Staubli VAL3: SocketMove.dtx

mdesc mNomSpeed
string sGetStr
sio sS = {link=Socket\ss}
string sBuff
trsf trTrsf
trsf trPara
bool bRes
mdesc mRun
pointRx pPrun = {fatherId=world[0]}
tool tTool = {z=100, fatherId=flange[0], ioLink=valve1}
jointRx jrun
pointRx pPMovec = {fatherId=world[0]}
pointRx pCurrent = {fatherId=world[0]}
trsf trSafety = {x=924.6, y=357.15, z=-147.43, ry=-180, rz=-1.37}
bool bOverRun
num nRobotSpeed
